// TwinCAT 3 PLC project Fermenter
// ProgramVersion: 3.1.4023.0
// libraries:
//   Tc2_Standard, * (Beckhoff Automation GmbH)
//   Tc2_System, * (Beckhoff Automation GmbH)
//   Tc3_Module, * (Beckhoff Automation GmbH)
//   VisuDialogs, * (System)
//   VisuSymbols,3.5.10.0,System
// project tree:
//   / GlobalTextList.TcGTLO, PlcTask.TcTTO, Visualization Manager.TcVMO (not stored)
//   POUs/ LDD.TcPOU, MAIN.TcPOU, SFC.TcPOU
//   VISUs/ FermenterControl.TcVIS
// real-time tasks:
//   TASK PlcTask: cycle T#10ms, priority 20, ADS port 350
//   TASK PlcTask1: cycle T#10ms, priority 21, ADS port 351

CONFIGURATION Fermenter
    RESOURCE PLC ON TwinCAT3
        TASK PlcTask(INTERVAL := T#10ms, PRIORITY := 21);
        PROGRAM MAIN WITH PlcTask : MAIN;
    END_RESOURCE
END_CONFIGURATION

// ---- POUs/MAIN.TcPOU
PROGRAM MAIN
VAR
END_VAR

SFC();

END_PROGRAM

// ---- POUs/SFC.TcPOU
PROGRAM SFC
VAR
	Run: BOOL;
	After15s: BOOL;
	Finished: BOOL;
	SteamIn: BOOL;
	Drain: BOOL;
	WaterIn: BOOL;
	GlycolIn: BOOL;
	GlycolOut: BOOL;
	Temp: REAL;
	FlushTimer: TON;
	Temp_GE_70: BOOL;
	Temp_LE_4: BOOL;
	Temp_LT_20: BOOL;
END_VAR

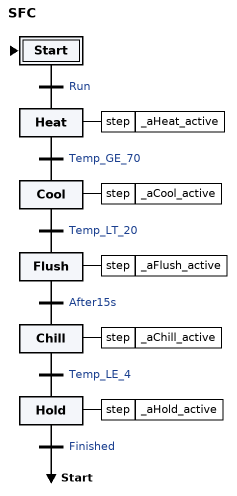
INITIAL_STEP Start:
END_STEP
TRANSITION FROM Start TO Heat
    := Run;
END_TRANSITION
STEP Heat:
    _aHeat_active(N);  // step action
END_STEP
TRANSITION FROM Heat TO Cool
    := Temp_GE_70;
END_TRANSITION
STEP Cool:
    _aCool_active(N);  // step action
END_STEP
TRANSITION FROM Cool TO Flush
    := Temp_LT_20;
END_TRANSITION
STEP Flush:
    _aFlush_active(N);  // step action
END_STEP
TRANSITION FROM Flush TO Chill
    := After15s;
END_TRANSITION
STEP Chill:
    _aChill_active(N);  // step action
END_STEP
TRANSITION FROM Chill TO Hold
    := Temp_LE_4;
END_TRANSITION
STEP Hold:
    _aHold_active(N);  // step action
END_STEP
TRANSITION FROM Hold TO Start
    := Finished;
END_TRANSITION

ACTION _aChill_active:
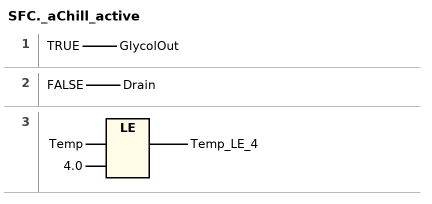
// NETWORK 1
GlycolOut := TRUE;

// NETWORK 2
Drain := FALSE;

// NETWORK 3
Temp_LE_4 := Temp <= 4.0;
END_ACTION

ACTION _aCool_active:
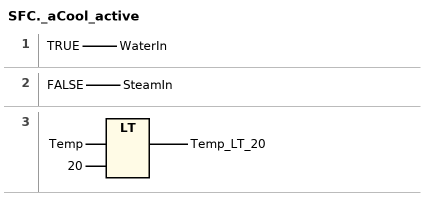
// NETWORK 1
WaterIn := TRUE;

// NETWORK 2
SteamIn := FALSE;

// NETWORK 3
Temp_LT_20 := Temp < 20;
END_ACTION

ACTION _aFlush_active:
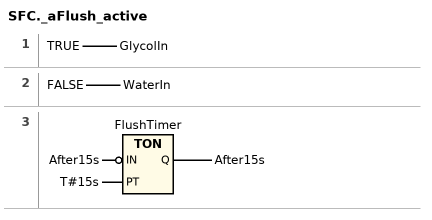
// NETWORK 1
GlycolIn := TRUE;

// NETWORK 2
WaterIn := FALSE;

// NETWORK 3
FlushTimer(IN := NOT After15s, PT := T#15s); // TON
After15s := FlushTimer.Q;
END_ACTION

ACTION _aHeat_active:
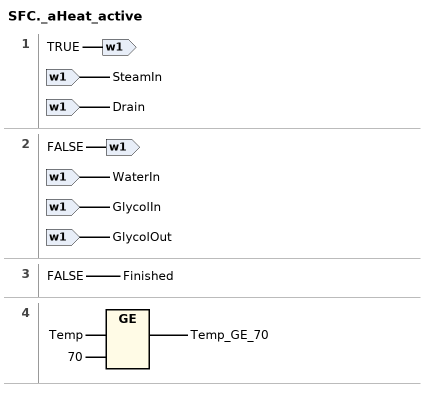
// NETWORK 1
SteamIn := TRUE;
Drain := TRUE;

// NETWORK 2
WaterIn := FALSE;
GlycolIn := FALSE;
GlycolOut := FALSE;

// NETWORK 3
Finished := FALSE;

// NETWORK 4
Temp_GE_70 := Temp >= 70;
END_ACTION

ACTION _aHold_active:
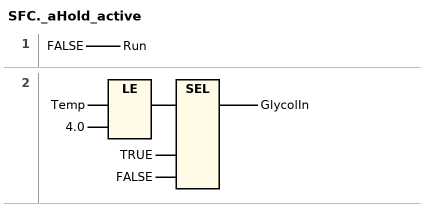
// NETWORK 1
Run := FALSE;

// NETWORK 2
GlycolIn := SEL(Temp <= 4.0, TRUE, FALSE);
END_ACTION

END_PROGRAM

// ---- POUs/LDD.TcPOU
PROGRAM LDD
VAR
	Start: BOOL:= TRUE;
	Heat: BOOL;
	Cool: BOOL;
	Flush: BOOL;
	Chill: BOOL;
	Hold: BOOL;
	Con1: BOOL;
	Run: BOOL;
	SteamIn: BOOL;
	Drain: BOOL;
	Temp: REAL;
	WaterIn: BOOL;
	GlycolIn: BOOL;
	GlycolOut: BOOL;
	FlushTimer: TON;
	Finished: BOOL;
END_VAR
VAR // added by the converter: edge detectors and wires of the graphical bodies
    _w1, _w2, _w3, _w4, _w5, _w6, _w7, _w8, _w9, _w10 : BOOL;
END_VAR

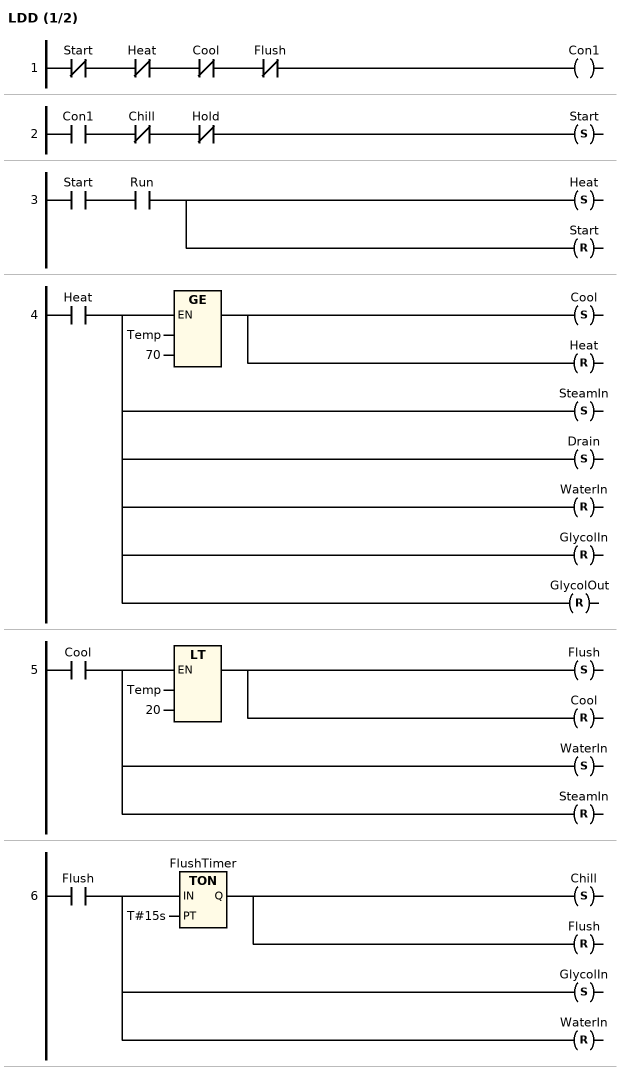
// NETWORK 1
Con1 := NOT Start AND NOT Heat AND NOT Cool AND NOT Flush;

// NETWORK 2
Start S= Con1 AND NOT Chill AND NOT Hold;

// NETWORK 3
_w1 := Start AND Run;
Heat S= _w1;
Start R= _w1;

// NETWORK 4
_w2 := Heat;
_w3 := _w2 AND Temp >= 70;
Cool S= _w3;
Heat R= _w3;
SteamIn S= _w2;
Drain S= _w2;
WaterIn R= _w2;
GlycolIn R= _w2;
GlycolOut R= _w2;

// NETWORK 5
_w4 := Cool;
_w5 := _w4 AND Temp < 20;
Flush S= _w5;
Cool R= _w5;
WaterIn S= _w4;
SteamIn R= _w4;

// NETWORK 6
_w6 := Flush;
FlushTimer(IN := _w6, PT := T#15s); // TON
Chill S= FlushTimer.Q;
Flush R= FlushTimer.Q;
GlycolIn S= _w6;
WaterIn R= _w6;

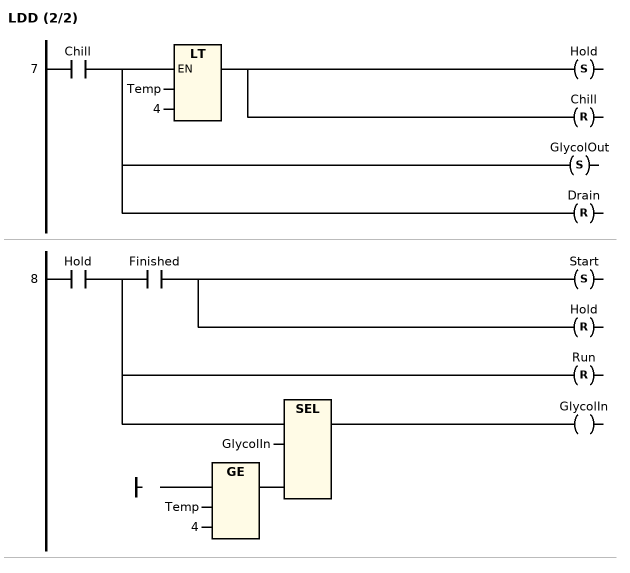
// NETWORK 7
_w7 := Chill;
_w8 := _w7 AND Temp < 4;
Hold S= _w8;
Chill R= _w8;
GlycolOut S= _w7;
Drain R= _w7;

// NETWORK 8
_w9 := Hold;
_w10 := _w9 AND Finished;
Start S= _w10;
Hold R= _w10;
Run R= _w9;
GlycolIn := SEL(_w9, GlycolIn, Temp >= 4);

END_PROGRAM

// ---- GlobalTextList.TcGTLO
TEXTLIST GlobalTextList
  115 = 'Drain'
  170 = 'Glycol In'
  111 = 'Glycol Out'
  932 = 'Steam In'
  649 = 'Water In'
END_TEXTLIST

// ---- VISUs/FermenterControl.TcVIS
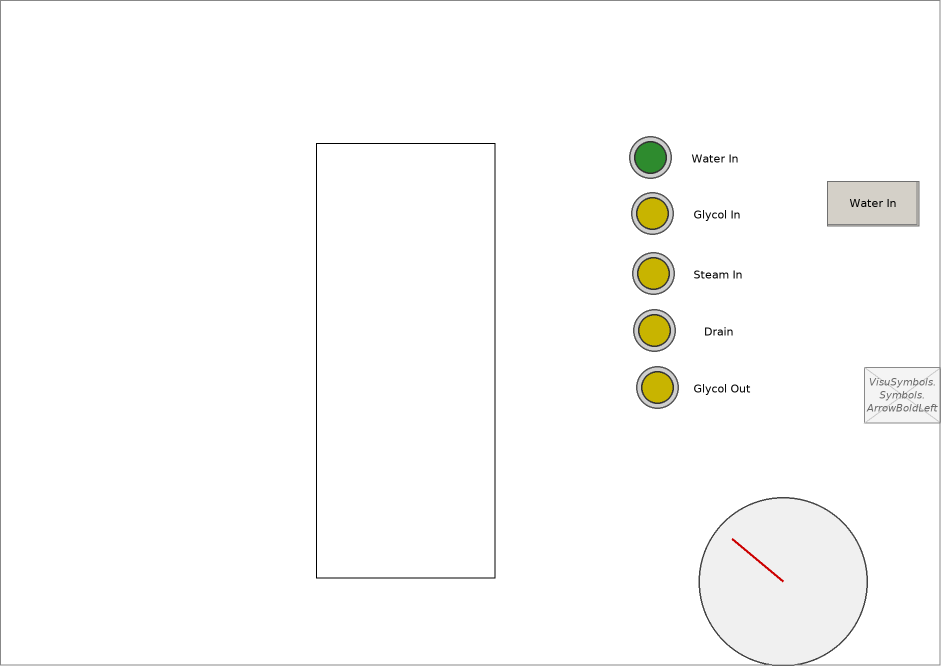
VISUALIZATION FermenterControl  // 941x666
    Rectangle (316,143 179x435)
    Lamp1 (624,133 53x49), variable: SFC.WaterIn, style: Lamp-Lamp1-Green
    Label (677,145 76x28), "Water In"
    Label (679,201 76x28), "Glycol In"
    Lamp1 (626,189 53x49), variable: SFC.GlycolIn, style: Lamp-Lamp1-Yellow
    Label (680,261 76x28), "Steam In"
    Lamp1 (627,249 53x49), variable: SFC.SteamIn, style: Lamp-Lamp1-Yellow
    Label (681,318 76x28), "Drain"
    Lamp1 (628,306 53x49), variable: SFC.Drain, style: Lamp-Lamp1-Yellow
    Label (684,375 76x28), "Glycol Out"
    Lamp1 (631,363 53x49), variable: SFC.GlycolOut, style: Lamp-Lamp1-Yellow
    Meter180 (651,497 264x169), value: SFC.Temp, style: Meter-Meter180-Gray, scale format: %.1f, scale 0..100
    Button (827,181 92x45), "Water In"
        OnMouseUp: toggle SFC.WaterIn
    Image (864,367 77x56), image: VisuSymbols.Symbols.ArrowBoldLeft
END_VISUALIZATION
